PROGRAM MAIN
VAR
	bBrowserStart: BOOL;
END_VAR

AlarmSample();// Пример работы с авариями

TrendSample();

END_PROGRAM

(* stored: Version 1.1.0.1, ProductVersion 3.1.4024.10
   POU MAIN: Id {4c756481-7ec3-4e41-a368-ed1e2246c441}, SpecialFunc None *)
